(* IEC 61131-3 sources: ICSML/Codesys_V3/Function Blocks/Sigmoid_L.pou, 1 file *)

(* ---- Sigmoid_L.pou ---- *)
(*#-#-#-#-#-#-#-#-#-#---Declaration---#-#-#-#-#-#-#-#-#-#-#-#-#*)

(*
	Sigmoid Activation Layer
*)
FUNCTION_BLOCK PUBLIC Sigmoid_L IMPLEMENTS Activation
VAR
	// Input and Output dataMem variables
	input_i: dataMem;
	output_i: dataMem;
END_VAR
(*#-#-#-#-#-#-#-#-#-#---Implementation---#-#-#-#-#-#-#-#-#-#-#-#-#*)
